// TIA Portal V19 export
DATA_BLOCK "AI SCALING DB"   // DB5
{ S7_Optimized_Access := 'TRUE' }
// stored: MemoryReserve 100
   VAR RETAIN
      MIN : Struct
         "LOAD CELL- MFG" : Real;
         "LOAD CELL- PREMIXING" : Real;
         "LOAD CELL- SUGAR" : Real;
         "LOAD CELL- STORAGE-1" : Real;
         "LOAD CELL- STORAGE-2" : Real;
         "CONDUCTIVITY METER" : Real;
         "TEMP.SENSOR- MFG INLET" : Real;
         "TEMP.SENSOR- MFG OUTLET" : Real;
         "TEMP.SENSOR- PREMIXING INLET" : Real;
         "TEMP.SENSOR- PREMIXING OUTLET" : Real;
         "TEMP.SENSOR- SUGAR INLET" : Real;
         "TEMP.SENSOR- SUGAR OUTLET" : Real;
         "TEMP.SENSOR- CIP" : Real;
         "PRESSURE TRANSMTER- MFG" : Real;
         "PRESSURE TRANSMTER- SUGAR" : Real;
         "VACUUME TRANSMTER- MFG" : Real;
         "VACUUME TRANSMTER- SUGAR" : Real;
         "VACUUME TRANSMTER- PREMIXING" : Real;
         "AI SPARE_1" : Real;
         "AI SPARE_2" : Real;
         "AI SPARE_3" : Real;
         "AI SPARE_4" : Real;
         "AI SPARE_5" : Real;
         "AI SPARE_6" : Real;
      END_STRUCT;
      MAX : Struct
         "LOAD CELL- MFG" : Real;
         "LOAD CELL- PREMIXING" : Real;
         "LOAD CELL- SUGAR" : Real;
         "LOAD CELL- STORAGE-1" : Real;
         "LOAD CELL- STORAGE-2" : Real;
         "CONDUCTIVITY METER" : Real;
         "TEMP.SENSOR- MFG INLET" : Real;
         "TEMP.SENSOR- MFG OUTLET" : Real;
         "TEMP.SENSOR- PREMIXING INLET" : Real;
         "TEMP.SENSOR- PREMIXING OUTLET" : Real;
         "TEMP.SENSOR- SUGAR INLET" : Real;
         "TEMP.SENSOR- SUGAR OUTLET" : Real;
         "TEMP.SENSOR- CIP" : Real;
         "PRESSURE TRANSMTER- MFG" : Real;
         "PRESSURE TRANSMTER- SUGAR" : Real;
         "VACUUME TRANSMTER- MFG" : Real;
         "VACUUME TRANSMTER- SUGAR" : Real;
         "VACUUME TRANSMTER- PREMIXING" : Real;
         "AI SPARE_1" : Real;
         "AI SPARE_2" : Real;
         "AI SPARE_3" : Real;
         "AI SPARE_4" : Real;
         "AI SPARE_5" : Real;
         "AI SPARE_6" : Real;
      END_STRUCT;
   END_VAR
   VAR
      PV : Struct
         "LOAD CELL- MFG" : Real;
         "LOAD CELL- PREMIXING" : Real;
         "LOAD CELL- SUGAR" : Real;
         "LOAD CELL- STORAGE-1" : Real;
         "LOAD CELL- STORAGE-2" : Real;
         "CONDUCTIVITY METER" : Real;
         "TEMP.SENSOR- MFG INLET" : Real;
         "TEMP.SENSOR- MFG OUTLET" : Real;
         "TEMP.SENSOR- PREMIXING INLET" : Real;
         "TEMP.SENSOR- PREMIXING OUTLET" : Real;
         "TEMP.SENSOR- SUGAR INLET" : Real;
         "TEMP.SENSOR- SUGAR OUTLET" : Real;
         "TEMP.SENSOR- CIP" : Real;
         "PRESSURE TRANSMTER- MFG" : Real;
         "PRESSURE TRANSMTER- SUGAR" : Real;
         "VACUUME TRANSMTER- MFG" : Real;
         "VACUUME TRANSMTER- SUGAR" : Real;
         "VACUUME TRANSMTER- PREMIXING" : Real;
         "AI SPARE_1" : Real;
         "AI SPARE_2" : Real;
         "AI SPARE_3" : Real;
         "AI SPARE_4" : Real;
         "AI SPARE_5" : Real;
         "AI SPARE_6" : Real;
      END_STRUCT;
   END_VAR
BEGIN
END_DATA_BLOCK
